(* IEC 61131-3 sources: simatic-ax-robotcontroller/src, 4 files *)

(* ---- Example.st ---- *)
NAMESPACE Simatic.Ax.DemoLibrary
    CLASS ExampleClass
        VAR PUBLIC

        END_VAR
        VAR PROTECTED
            _value : DINT;
        END_VAR

        //Next step: Generate Loadable to perform download to PLC

    END_CLASS
END_NAMESPACE

(* ---- WrapperFB.st ---- *)
NAMESPACE Simatic.Ax.DemoLibrary
    FUNCTION_BLOCK EnableRobotFB
        VAR_INPUT
            RobotRequest : BOOL;
            RobotBusy : Bool;
        END_VAR
        VAR_OUTPUT
            RobotEnable : Bool;
        END_VAR
        VAR
           _inst : ExampleClass;
        END_VAR

        RobotEnable := FALSE ;
        IF RobotRequest AND NOT RobotBusy THEN
            RobotEnable := TRUE;
        END_IF;
        //_inst.RunCyclic();

    END_FUNCTION_BLOCK
END_NAMESPACE

(* ---- configuration.st ---- *)
CONFIGURATION MyConfiguration
    TASK Main(Interval := T#1000ms, Priority := 1);
    PROGRAM P1 WITH Main: MyProgram;

    VAR_GLOBAL
        In AT %IW0 : INT;
        Out AT %QW2 : INT;
        toggle : BOOL;
        output_signal AT %Q0.1 : BOOL;
        count_value : LINT;
    END_VAR
END_CONFIGURATION

(* ---- program.st ---- *)
USING System.Counters;

PROGRAM MyProgram

    VAR_EXTERNAL
        In : INT;
        Out : INT;
        toggle : BOOL;
        output_signal: BOOL;
        count_value : LINT;

    END_VAR

    VAR
        count : CounterUp := (presetValue := 5);
    END_VAR

    Out := In;
    toggle := NOT toggle;
    count(up := toggle);
    output_signal := count.presetReached;
    count_value := count.value;
    count.reset := count_value >= 10;
    // to be done here:
    // Implement OPC Server
    //apax oscr interface install opcinterface.yml -t targetIP

    // OPC Server provides variables similar to MoPaHyb Interface
    // Implement State Manager similar to MoPaHyb Interface (see RPI implementation as reference) using simatic-ax\statemachine package from github
    // Implement Handshake with robot
    // testings
    ;
END_PROGRAM
